TYPE ST_LabelerRecipe :
	STRUCT
		Length				: LREAL;
//		LeftAxis			: ST_AxisRecipe;
//		RightAxis			: ST_AxisRecipe;
		CylinderExtendTime	: LREAL;
		CylinderRetractTime : LREAL;
	END_STRUCT
END_TYPE

(* stored: Version 1.1.0.1, ProductVersion 3.1.4024.15
   DUT ST_LabelerRecipe: Id {b481ce3f-8f0e-45c8-a330-fd8874c99800} *)
